FUNCTION_BLOCK my_sensor2 (* Composite Function Block Type *)
  (* Standard: 61499-2 *)
  (* Version 0.2, 2003-12-05, JHC, Rockwell Automation, Renamed from NEWCOMPFB. *)
  (* Version 0.1, 2002-01-08, JHC, Rockwell Automation, Added DLY FB as example. *)
  (* Version 0.0, 2000-05-27, JHC, Rockwell Automation *)
  (* Compiler header: package fb.rt.pnp; *)
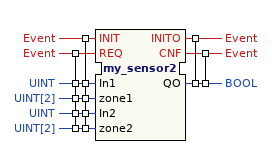
  EVENT_INPUT
    INIT WITH In1, zone1, In2, zone2; (* Initialization Request *)
    REQ WITH In1, zone1, In2, zone2; (* Normal Execution Request *)
  END_EVENT
  EVENT_OUTPUT
    INITO WITH QO; (* Initialization Confirm *)
    CNF WITH QO; (* Execution Confirmation *)
  END_EVENT
  VAR_INPUT
    In1 : UINT;
    zone1 : ARRAY [0..1] OF UINT;
    In2 : UINT;
    zone2 : ARRAY [0..1] OF UINT;
  END_VAR
  VAR_OUTPUT
    QO : BOOL; (* Output event qualifier *)
  END_VAR
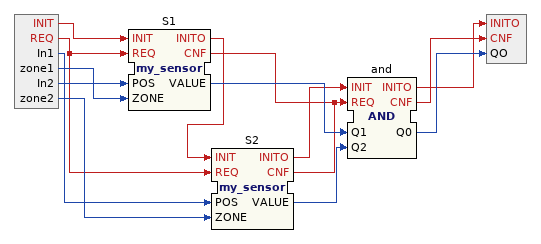
  FBS
    S1 : my_sensor;
    S2 : my_sensor;
    and : AND;
  END_FBS
  EVENT_CONNECTIONS
    INIT TO S1.INIT;
    S1.INITO TO S2.INIT;
    REQ TO S1.REQ;
    S2.INITO TO and.INIT;
    S1.CNF TO and.REQ;
    S2.CNF TO and.REQ;
    and.INITO TO INITO;
    and.CNF TO CNF;
    REQ TO S2.REQ;
  END_CONNECTIONS
  DATA_CONNECTIONS
    In1 TO S1.POS;
    zone1 TO S1.ZONE;
    In2 TO S2.POS;
    zone2 TO S2.ZONE;
    S1.VALUE TO and.Q1;
    S2.VALUE TO and.Q2;
    and.Q0 TO QO;
  END_CONNECTIONS
END_FUNCTION_BLOCK
